{attribute 'linkalways'} 
{attribute 'no_explicit_call' := 'This FB is a CLASS and must be accessed using methods or properties'}
{attribute 'enable_dynamic_creation'}
FUNCTION_BLOCK Node_F_VN_FillContainer_TcVnRectangle_DINT EXTENDS VisionNode
VAR
    ipContainer : _ITcVnContainer;
    stValue : _TcVnRectangle_DINT;
    hrPrev : _HRESULT(S_OK);
    hresult : _HRESULT(S_OK);
END_VAR

METHOD PUBLIC  Clone : I_Node
VAR
    pNode : POINTER TO Node_F_VN_FillContainer_TcVnRectangle_DINT;
END_VAR
pNode := __NEW(Node_F_VN_FillContainer_TcVnRectangle_DINT);
Clone := pNode^;
END_METHOD

METHOD FB_init : BOOL
VAR_INPUT
    bInitRetains : BOOL; // if TRUE, the retain variables are initialized (warm start / cold start)
    bInCopyCode : BOOL;  // if TRUE, the instance afterwards gets moved into the copy code (online change)
END_VAR
AddInput('ipContainer', ipContainer);
AddInput('stValue', stValue);
AddInput('hrPrev', hrPrev);
AddOutput('ipContainer', ipContainer);
AddOutput('hresult',hresult);
END_METHOD

METHOD PROTECTED OnExecute : HRESULT
hresult.Value := F_VN_FillContainer_TcVnRectangle_DINT(
    ipContainer := ipContainer.Value,
    stValue := stValue.Value,
    hrPrev:= hrPrev.Value);
END_METHOD

METHOD PUBLIC PreExecutionCheck
VAR_INPUT
    Check : I_PreExecutionChecks;
END_VAR
Check.IsTrue(ipContainer.IsValid, 'ipContainer must be a valid container');
END_METHOD

END_FUNCTION_BLOCK

(* stored: Version 1.1.0.1, ProductVersion 3.1.4024.13
   POU Node_F_VN_FillContainer_TcVnRectangle_DINT: Id {c9431519-0043-4d9e-93e7-2533f1d39043}, SpecialFunc None
   Folder Constructor: Id {68ba18c9-e434-42e2-b19b-b61ee8c9c90f}
   Method Clone: Id {8925083f-ba1f-4123-b65d-8c46a2e04856}
   Method FB_init: Id {c212c615-c66e-4067-85b6-7b66c3e97ba9}
   Method OnExecute: Id {6e6773e7-d807-4a26-86b0-b9441e07009f}
   Method PreExecutionCheck: Id {74ed8014-327b-46e9-b22f-655d1dd1c3e2} *)
